{attribute 'GeneratedUsingTerminal: EPP6228-0022-0016'}
{attribute addProperty BoxType "EPP6228-0022-0016"}
{attribute addProperty Id "DeviceState_InputsDeviceState_Inputs_C7251DC98"}
{attribute addProperty CRC "3106540906"}
{attribute addProperty Size "8"}
TYPE Module_2_DeviceState_Inputs_B92A0D6A :
STRUCT
	{attribute addProperty Name "DeviceState_Inputs"}
	DeviceState_Inputs  : DeviceState_Inputs_C7251DC9;
END_STRUCT
END_TYPE

(* stored: Version 1.2.0.0, ProductVersion 3.1.4024.9
   DUT Module_2_DeviceState_Inputs_B92A0D6A: Id {6d21e9b9-7898-4517-8cef-bcdfbb4fb2e8} *)
